(* CoDeSys 2.3 export: SELECTORSUBSTATUS.EXP *)

(* Data type in ENUM *)
TYPE SelectorSubStatus : (SelectorSubStatusNormal:=0, SelectorSubStatusChangePos, SelectorSubStatusRefStopped, SelectorSubStatusRefAlarm,
								SelectorSubStatusAlarm, SelectorSubStatusTimeout, SelectorSubStatusConfErr, SelectorSubStatusUnknownCommand,
								SelectorSubStatusBadCommandParameter);
END_TYPE
